Staubli VAL3: resetLatch.pgx

public program resetLatch()
begin
  bPartLatched=false
end
